% RSLogix 500 project Smart Pedestrian Crossing Controller using Allen-Bradley PLC.RSS, saved by version 8.30.00.16 %
PROJECT "UNTITLED"    % processor: Bul.1763 MicroLogix 1100 Series B %

PROGRAM FILES
  LAD 2   40 rungs

DATA FILES
  O0 OUTPUT  4 elements
  I1 INPUT  6 elements
  S2 STATUS  66 elements
  B3 BINARY  2 elements
  T4 TIMER  7 elements
  C5 COUNTER  1 elements
  R6 CONTROL  1 elements
  N7 INTEGER  1 elements
  F8 FLOAT  1 elements

LADDER 2
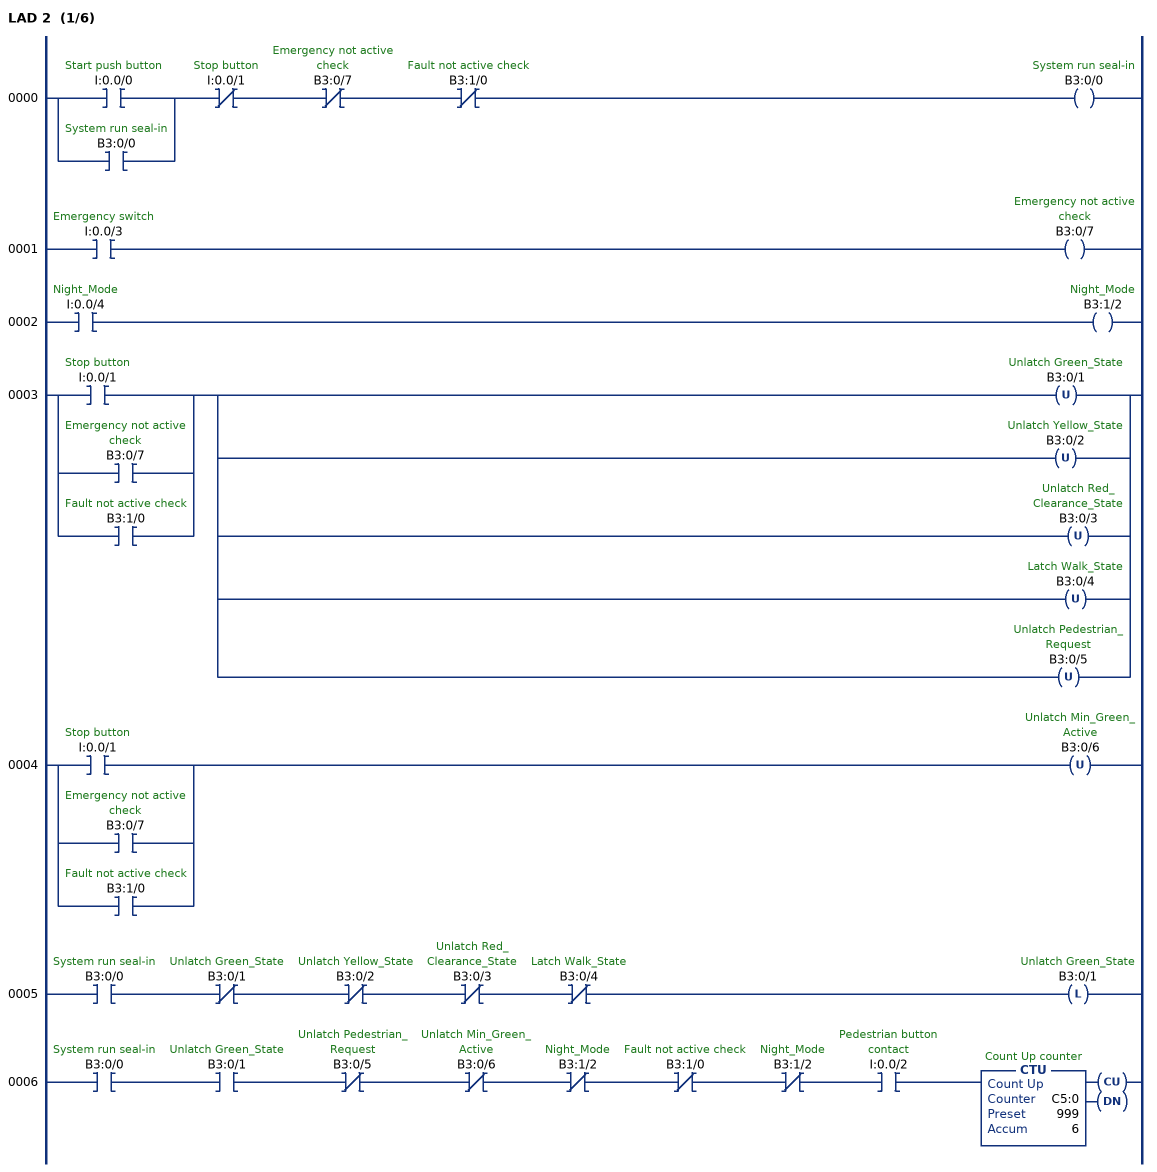
% Rung: 0 %
SOR BST XIC I:0.0/0 NXB XIC B3:0/0 BND XIO I:0.0/1 XIO B3:0/7 XIO B3:1/0 OTE B3:0/0 EOR
%   I:0.0/0  "Start push button" %
%   B3:0/0  "System run seal-in" %
%   I:0.0/1  "Stop button" %
%   B3:0/7  "Emergency not active check" %
%   B3:1/0  "Fault not active check" %
% Rung: 1 %
SOR XIC I:0.0/3 OTE B3:0/7 EOR
%   I:0.0/3  "Emergency switch" %
%   B3:0/7  "Emergency not active check" %
%   OTE B3:0/7  "Emergency_Mode Active" %
% Rung: 2 %
SOR XIC I:0.0/4 OTE B3:1/2 EOR
%   I:0.0/4  "Night_Mode" %
%   B3:1/2  "Night_Mode" %
% Rung: 3 %
SOR BST XIC I:0.0/1 NXB BST XIC B3:0/7 NXB XIC B3:1/0 BND BND BST OTU B3:0/1 NXB BST OTU B3:0/2 NXB BST OTU B3:0/3 NXB BST OTU B3:0/4 NXB OTU B3:0/5 BND BND BND BND EOR
%   I:0.0/1  "Stop button" %
%   B3:0/7  "Emergency not active check" %
%   XIC B3:0/7  "Emergency_Mode contact" %
%   B3:1/0  "Fault not active check" %
%   XIC B3:1/0  "Fault contact" %
%   B3:0/1  "Unlatch Green_State" %
%   B3:0/2  "Unlatch Yellow_State" %
%   B3:0/3  "Unlatch Red_Clearance_State" %
%   B3:0/4  "Latch Walk_State" %
%   OTU B3:0/4  "Unlatch Walk_State" %
%   B3:0/5  "Unlatch Pedestrian_Request" %
% Rung: 4 %
SOR BST XIC I:0.0/1 NXB BST XIC B3:0/7 NXB XIC B3:1/0 BND BND OTU B3:0/6 EOR
%   I:0.0/1  "Stop button" %
%   B3:0/7  "Emergency not active check" %
%   XIC B3:0/7  "Emergency_Mode contact" %
%   B3:1/0  "Fault not active check" %
%   XIC B3:1/0  "Fault contact" %
%   B3:0/6  "Unlatch Min_Green_Active" %
% Rung: 5 %
SOR XIC B3:0/0 XIO B3:0/1 XIO B3:0/2 XIO B3:0/3 XIO B3:0/4 OTL B3:0/1 EOR
%   B3:0/0  "System run seal-in" %
%   B3:0/1  "Unlatch Green_State" %
%   XIO B3:0/1  "Green_State not active" %
%   B3:0/2  "Unlatch Yellow_State" %
%   XIO B3:0/2  "Yellow_State not active" %
%   B3:0/3  "Unlatch Red_Clearance_State" %
%   XIO B3:0/3  "Red_Clearance_State not active contact" %
%   B3:0/4  "Latch Walk_State" %
%   XIO B3:0/4  "Walk_State not active" %
%   OTL B3:0/1  "Latch Green_State" %
% Rung: 6 %
SOR XIC B3:0/0 XIC B3:0/1 XIO B3:0/5 XIO B3:0/6 XIO B3:1/2 XIO B3:1/0 XIO B3:1/2 XIC I:0.0/2 CTU C5:0 999 6 EOR
%   B3:0/0  "System run seal-in" %
%   B3:0/1  "Unlatch Green_State" %
%   XIC B3:0/1  "Green_State contact" %
%   B3:0/5  "Unlatch Pedestrian_Request" %
%   XIO B3:0/5  "No request already stored" %
%   B3:0/6  "Unlatch Min_Green_Active" %
%   XIO B3:0/6  "Minimum green not active" %
%   B3:1/2  "Night_Mode" %
%   B3:1/0  "Fault not active check" %
%   I:0.0/2  "Pedestrian button contact" %
%   C5:0  "Count Up counter" %

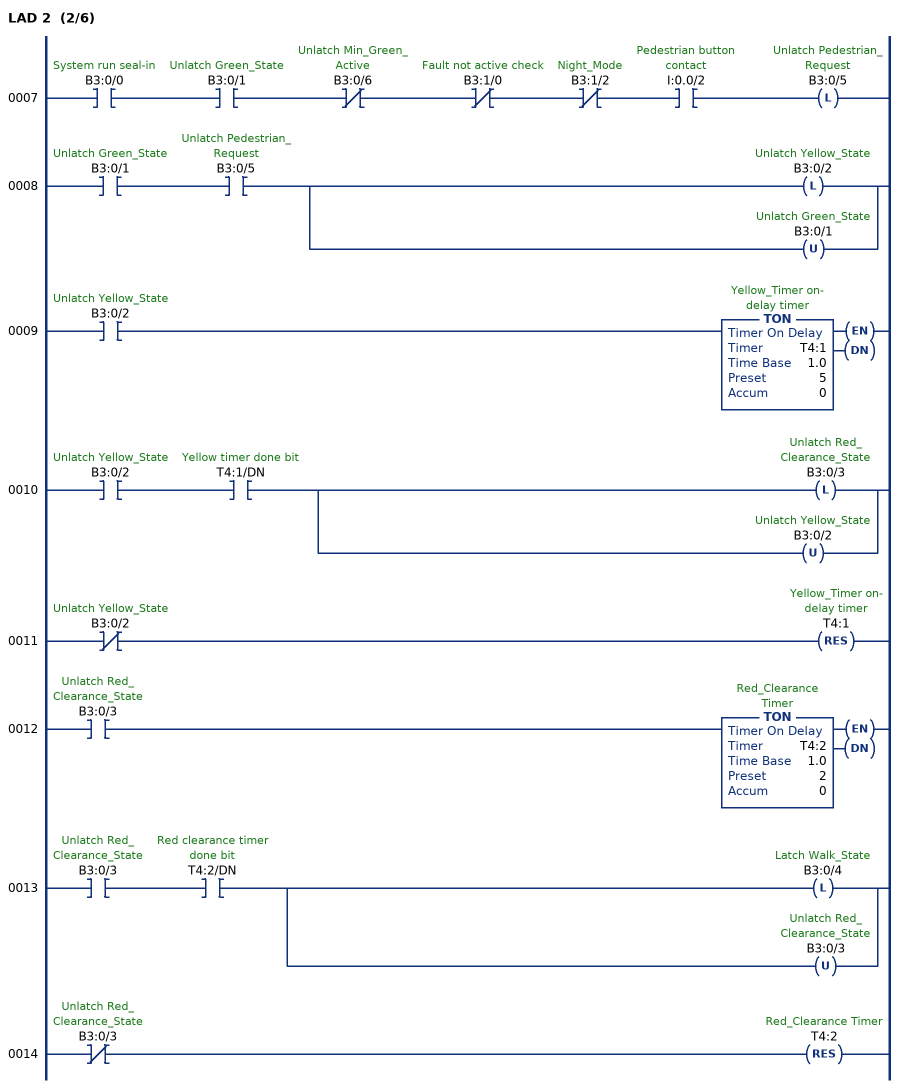
% Rung: 7 %
SOR XIC B3:0/0 XIC B3:0/1 XIO B3:0/6 XIO B3:1/0 XIO B3:1/2 XIC I:0.0/2 OTL B3:0/5 EOR
%   B3:0/0  "System run seal-in" %
%   B3:0/1  "Unlatch Green_State" %
%   XIC B3:0/1  "Green_State contact" %
%   B3:0/6  "Unlatch Min_Green_Active" %
%   XIO B3:0/6  "Minimum green not active" %
%   B3:1/0  "Fault not active check" %
%   B3:1/2  "Night_Mode" %
%   I:0.0/2  "Pedestrian button contact" %
%   B3:0/5  "Unlatch Pedestrian_Request" %
%   OTL B3:0/5  "Latch Pedestrian_Request" %
% Rung: 8 %
SOR XIC B3:0/1 XIC B3:0/5 BST OTL B3:0/2 NXB OTU B3:0/1 BND EOR
%   B3:0/1  "Unlatch Green_State" %
%   XIC B3:0/1  "Green_State contact" %
%   B3:0/5  "Unlatch Pedestrian_Request" %
%   XIC B3:0/5  "Pedestrian_Request contact" %
%   B3:0/2  "Unlatch Yellow_State" %
%   OTL B3:0/2  "Latch Yellow_State" %
% Rung: 9 %
SOR XIC B3:0/2 TON T4:1 1.0 5 0 EOR
%   B3:0/2  "Unlatch Yellow_State" %
%   XIC B3:0/2  "Yellow_State contact" %
%   T4:1  "Yellow_Timer on- delay timer" %
% Rung: 10 %
SOR XIC B3:0/2 XIC T4:1/DN BST OTL B3:0/3 NXB OTU B3:0/2 BND EOR
%   B3:0/2  "Unlatch Yellow_State" %
%   XIC B3:0/2  "Yellow_State contact" %
%   T4:1/DN  "Yellow timer done bit" %
%   B3:0/3  "Unlatch Red_Clearance_State" %
%   OTL B3:0/3  "Latch Red_Clearance_State" %
% Rung: 11 %
SOR XIO B3:0/2 RES T4:1 EOR
%   B3:0/2  "Unlatch Yellow_State" %
%   XIO B3:0/2  "Yellow_State not active" %
%   T4:1  "Yellow_Timer on- delay timer" %
%   RES T4:1  "Reset Yellow_Timer" %
% Rung: 12 %
SOR XIC B3:0/3 TON T4:2 1.0 2 0 EOR
%   B3:0/3  "Unlatch Red_Clearance_State" %
%   XIC B3:0/3  "Red_Clearance_State contact" %
%   T4:2  "Red_Clearance Timer" %
% Rung: 13 %
SOR XIC B3:0/3 XIC T4:2/DN BST OTL B3:0/4 NXB OTU B3:0/3 BND EOR
%   B3:0/3  "Unlatch Red_Clearance_State" %
%   XIC B3:0/3  "Red_Clearance_State contact" %
%   T4:2/DN  "Red clearance timer done bit" %
%   B3:0/4  "Latch Walk_State" %
% Rung: 14 %
SOR XIO B3:0/3 RES T4:2 EOR
%   B3:0/3  "Unlatch Red_Clearance_State" %
%   XIO B3:0/3  "Red_Clearance_State not active contact" %
%   T4:2  "Red_Clearance Timer" %
%   RES T4:2  "Reset Red_Clearance_Timer" %

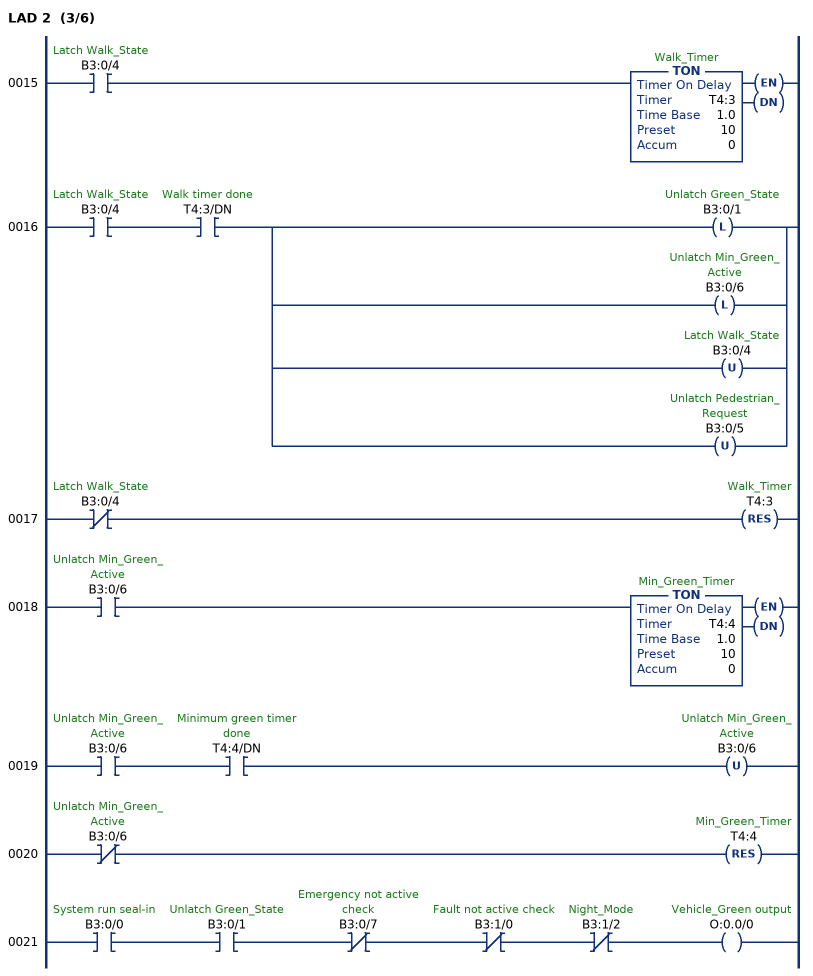
% Rung: 15 %
SOR XIC B3:0/4 TON T4:3 1.0 10 0 EOR
%   B3:0/4  "Latch Walk_State" %
%   XIC B3:0/4  "Walk_State contact" %
%   T4:3  "Walk_Timer" %
% Rung: 16 %
SOR XIC B3:0/4 XIC T4:3/DN BST OTL B3:0/1 NXB BST OTL B3:0/6 NXB BST OTU B3:0/4 NXB OTU B3:0/5 BND BND BND EOR
%   B3:0/4  "Latch Walk_State" %
%   XIC B3:0/4  "Walk_State contact" %
%   T4:3/DN  "Walk timer done" %
%   B3:0/1  "Unlatch Green_State" %
%   OTL B3:0/1  "Latch Green_State" %
%   B3:0/6  "Unlatch Min_Green_Active" %
%   OTL B3:0/6  "Latch Min_Green_Active" %
%   OTU B3:0/4  "Unlatch Walk_State" %
%   B3:0/5  "Unlatch Pedestrian_Request" %
% Rung: 17 %
SOR XIO B3:0/4 RES T4:3 EOR
%   B3:0/4  "Latch Walk_State" %
%   XIO B3:0/4  "Walk_State not active" %
%   T4:3  "Walk_Timer" %
%   RES T4:3  "Reset Walk_Timer" %
% Rung: 18 %
SOR XIC B3:0/6 TON T4:4 1.0 10 0 EOR
%   B3:0/6  "Unlatch Min_Green_Active" %
%   XIC B3:0/6  "Min_Green_Active contact" %
%   T4:4  "Min_Green_Timer" %
% Rung: 19 %
SOR XIC B3:0/6 XIC T4:4/DN OTU B3:0/6 EOR
%   B3:0/6  "Unlatch Min_Green_Active" %
%   XIC B3:0/6  "Min_Green_Active contact" %
%   T4:4/DN  "Minimum green timer done" %
% Rung: 20 %
SOR XIO B3:0/6 RES T4:4 EOR
%   B3:0/6  "Unlatch Min_Green_Active" %
%   XIO B3:0/6  "Minimum green not active" %
%   T4:4  "Min_Green_Timer" %
%   RES T4:4  "Reset Min_Green_Timer" %
% Rung: 21 %
SOR XIC B3:0/0 XIC B3:0/1 XIO B3:0/7 XIO B3:1/0 XIO B3:1/2 OTE O:0.0/0 EOR
%   B3:0/0  "System run seal-in" %
%   B3:0/1  "Unlatch Green_State" %
%   XIC B3:0/1  "Green_State contact" %
%   B3:0/7  "Emergency not active check" %
%   B3:1/0  "Fault not active check" %
%   B3:1/2  "Night_Mode" %
%   O:0.0/0  "Vehicle_Green output" %

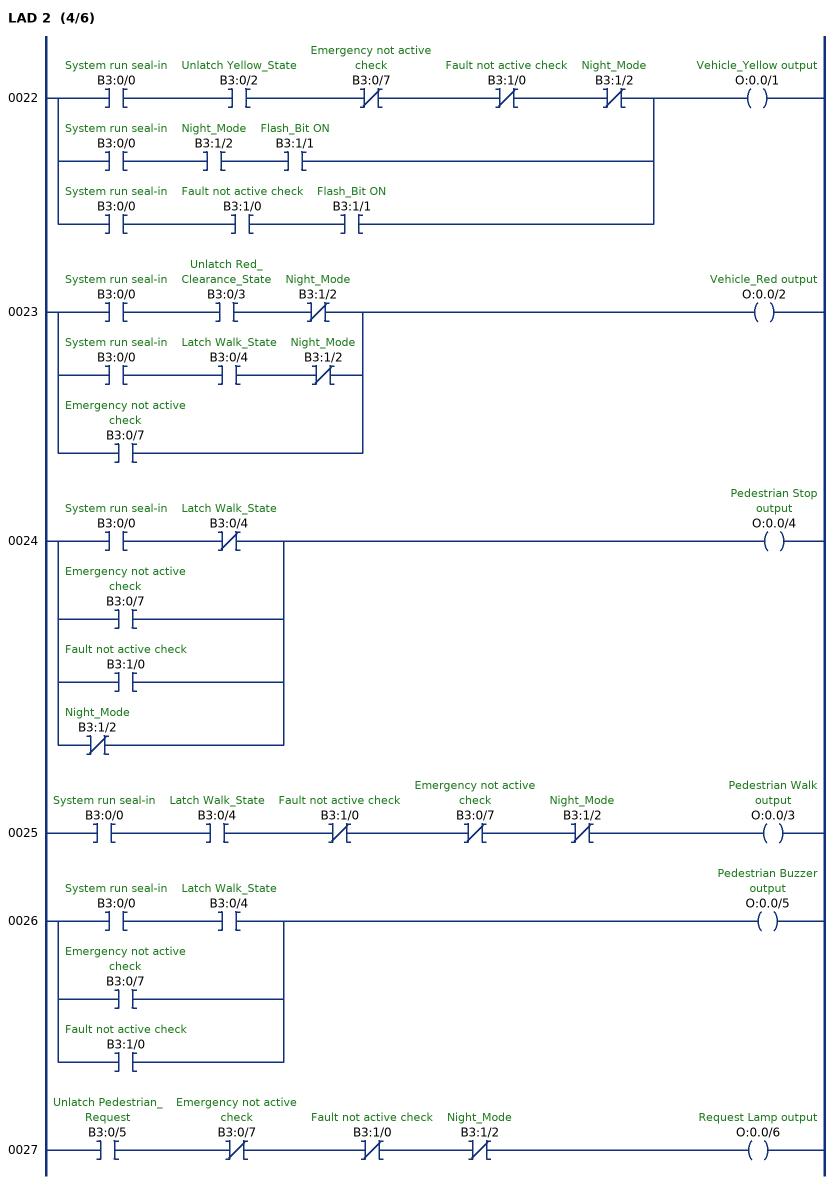
% Rung: 22 %
SOR BST XIC B3:0/0 XIC B3:0/2 XIO B3:0/7 XIO B3:1/0 XIO B3:1/2 NXB BST XIC B3:0/0 XIC B3:1/2 XIC B3:1/1 NXB XIC B3:0/0 XIC B3:1/0 XIC B3:1/1 BND BND OTE O:0.0/1 EOR
%   B3:0/0  "System run seal-in" %
%   B3:0/2  "Unlatch Yellow_State" %
%   XIC B3:0/2  "Yellow_State contact" %
%   B3:0/7  "Emergency not active check" %
%   B3:1/0  "Fault not active check" %
%   B3:1/2  "Night_Mode" %
%   B3:1/1  "Flash_Bit ON" %
%   XIC B3:1/0  "Fault contact" %
%   O:0.0/1  "Vehicle_Yellow output" %
% Rung: 23 %
SOR BST XIC B3:0/0 XIC B3:0/3 XIO B3:1/2 NXB BST XIC B3:0/0 XIC B3:0/4 XIO B3:1/2 NXB XIC B3:0/7 BND BND OTE O:0.0/2 EOR
%   B3:0/0  "System run seal-in" %
%   B3:0/3  "Unlatch Red_Clearance_State" %
%   XIC B3:0/3  "Red_Clearance_State contact" %
%   B3:1/2  "Night_Mode" %
%   B3:0/4  "Latch Walk_State" %
%   XIC B3:0/4  "Walk_State contact" %
%   B3:0/7  "Emergency not active check" %
%   XIC B3:0/7  "Emergency_Mode contact" %
%   O:0.0/2  "Vehicle_Red output" %
% Rung: 24 %
SOR BST XIC B3:0/0 XIO B3:0/4 NXB BST XIC B3:0/7 NXB BST XIC B3:1/0 NXB XIO B3:1/2 BND BND BND OTE O:0.0/4 EOR
%   B3:0/0  "System run seal-in" %
%   B3:0/4  "Latch Walk_State" %
%   XIO B3:0/4  "Walk_State not active" %
%   B3:0/7  "Emergency not active check" %
%   XIC B3:0/7  "Emergency_Mode contact" %
%   B3:1/0  "Fault not active check" %
%   XIC B3:1/0  "Fault contact" %
%   B3:1/2  "Night_Mode" %
%   O:0.0/4  "Pedestrian Stop output" %
% Rung: 25 %
SOR XIC B3:0/0 XIC B3:0/4 XIO B3:1/0 XIO B3:0/7 XIO B3:1/2 OTE O:0.0/3 EOR
%   B3:0/0  "System run seal-in" %
%   B3:0/4  "Latch Walk_State" %
%   XIC B3:0/4  "Walk_State contact" %
%   B3:1/0  "Fault not active check" %
%   B3:0/7  "Emergency not active check" %
%   B3:1/2  "Night_Mode" %
%   O:0.0/3  "Pedestrian Walk output" %
% Rung: 26 %
SOR BST XIC B3:0/0 XIC B3:0/4 NXB BST XIC B3:0/7 NXB XIC B3:1/0 BND BND OTE O:0.0/5 EOR
%   B3:0/0  "System run seal-in" %
%   B3:0/4  "Latch Walk_State" %
%   XIC B3:0/4  "Walk_State contact" %
%   B3:0/7  "Emergency not active check" %
%   XIC B3:0/7  "Emergency_Mode contact" %
%   B3:1/0  "Fault not active check" %
%   XIC B3:1/0  "Fault contact" %
%   O:0.0/5  "Pedestrian Buzzer output" %
% Rung: 27 %
SOR XIC B3:0/5 XIO B3:0/7 XIO B3:1/0 XIO B3:1/2 OTE O:0.0/6 EOR
%   B3:0/5  "Unlatch Pedestrian_Request" %
%   XIC B3:0/5  "Pedestrian_Request contact" %
%   B3:0/7  "Emergency not active check" %
%   B3:1/0  "Fault not active check" %
%   B3:1/2  "Night_Mode" %
%   O:0.0/6  "Request Lamp output" %

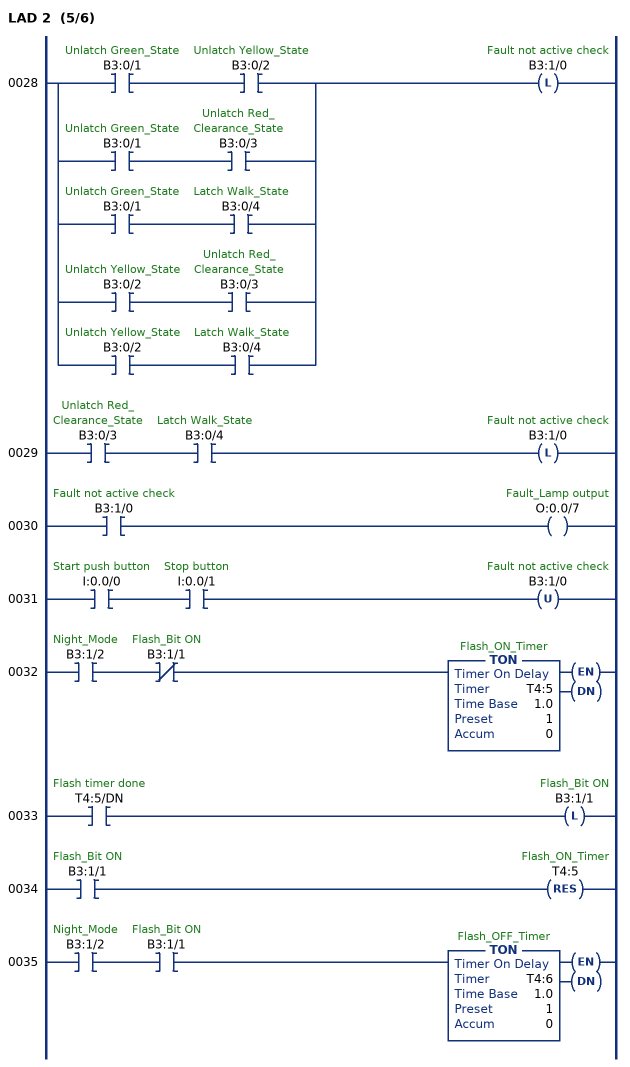
% Rung: 28 %
SOR BST XIC B3:0/1 XIC B3:0/2 NXB BST XIC B3:0/1 XIC B3:0/3 NXB BST XIC B3:0/1 XIC B3:0/4 NXB BST XIC B3:0/2 XIC B3:0/3 NXB XIC B3:0/2 XIC B3:0/4 BND BND BND BND OTL B3:1/0 EOR
%   B3:0/1  "Unlatch Green_State" %
%   XIC B3:0/1  "Green_State contact" %
%   B3:0/2  "Unlatch Yellow_State" %
%   XIC B3:0/2  "Yellow_State contact" %
%   B3:0/3  "Unlatch Red_Clearance_State" %
%   XIC B3:0/3  "Red_Clearance_State contact" %
%   B3:0/4  "Latch Walk_State" %
%   XIC B3:0/4  "Walk_State contact" %
%   B3:1/0  "Fault not active check" %
%   OTL B3:1/0  "Latch Fault bit" %
% Rung: 29 %
SOR XIC B3:0/3 XIC B3:0/4 OTL B3:1/0 EOR
%   B3:0/3  "Unlatch Red_Clearance_State" %
%   XIC B3:0/3  "Red_Clearance_State contact" %
%   B3:0/4  "Latch Walk_State" %
%   XIC B3:0/4  "Walk_State contact" %
%   B3:1/0  "Fault not active check" %
%   OTL B3:1/0  "Latch Fault bit" %
% Rung: 30 %
SOR XIC B3:1/0 OTE O:0.0/7 EOR
%   B3:1/0  "Fault not active check" %
%   XIC B3:1/0  "Fault contact" %
%   O:0.0/7  "Fault_Lamp output" %
% Rung: 31 %
SOR XIC I:0.0/0 XIC I:0.0/1 OTU B3:1/0 EOR
%   I:0.0/0  "Start push button" %
%   I:0.0/1  "Stop button" %
%   B3:1/0  "Fault not active check" %
%   OTU B3:1/0  "Unlatch Fault" %
% Rung: 32 %
SOR XIC B3:1/2 XIO B3:1/1 TON T4:5 1.0 1 0 EOR
%   B3:1/2  "Night_Mode" %
%   B3:1/1  "Flash_Bit ON" %
%   XIO B3:1/1  "Flash_Bit OFF" %
%   T4:5  "Flash_ON_Timer" %
% Rung: 33 %
SOR XIC T4:5/DN OTL B3:1/1 EOR
%   T4:5/DN  "Flash timer done" %
%   B3:1/1  "Flash_Bit ON" %
%   OTL B3:1/1  "Flash_Bit ON" %
% Rung: 34 %
SOR XIC B3:1/1 RES T4:5 EOR
%   B3:1/1  "Flash_Bit ON" %
%   T4:5  "Flash_ON_Timer" %
% Rung: 35 %
SOR XIC B3:1/2 XIC B3:1/1 TON T4:6 1.0 1 0 EOR
%   B3:1/2  "Night_Mode" %
%   B3:1/1  "Flash_Bit ON" %
%   T4:6  "Flash_OFF_Timer" %

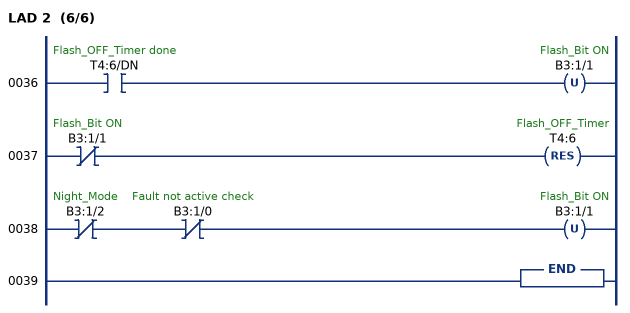
% Rung: 36 %
SOR XIC T4:6/DN OTU B3:1/1 EOR
%   T4:6/DN  "Flash_OFF_Timer done" %
%   B3:1/1  "Flash_Bit ON" %
% Rung: 37 %
SOR XIO B3:1/1 RES T4:6 EOR
%   B3:1/1  "Flash_Bit ON" %
%   XIO B3:1/1  "Flash_Bit OFF" %
%   T4:6  "Flash_OFF_Timer" %
% Rung: 38 %
SOR XIO B3:1/2 XIO B3:1/0 OTU B3:1/1 EOR
%   B3:1/2  "Night_Mode" %
%   B3:1/0  "Fault not active check" %
%   B3:1/1  "Flash_Bit ON" %
% Rung: 39 %
SOR END EOR

DATA TABLE (non-zero values as saved)
DATA T4
% .PRE .ACC %
% T4:1 % 5 0
% T4:2 % 2 0
% T4:3 % 10 0
% T4:4 % 10 0
% T4:5 % 1 0
% T4:6 % 1 0
DATA C5
% .PRE .ACC %
% C5:0 % 999 6
